FUNCTION_BLOCK CoolingNetwork
VAR_INPUT
	//feed temperature setpoint and system enabling
	fSetPoint_CN : REAL;
	fSetPoint_eChiller : REAL;
	fSetPoint_HVFAStorage : REAL;
	bLoading_HVFAStorage : BOOL;
	bSetStatusOn_eChiller : BOOL;
	bSetStatusOn_HeatPump : BOOL;
	bSetStatusOn_HVFAStorage : BOOL;	
END_VAR
VAR_OUTPUT
	//temperatures in buffer storage
	fTemperatureBufferStorage : REAL;
END_VAR
VAR
	//default parameters
	ST_HVFADefaultParameters : ST_HVFASystemDefaultParameters := (aSetPointLimitsTemperature:=[5,25]);

	//systems
	BufferStorage : FB_BufferStorage;
	eChillerSystem : FB_eChillerSystem;
	HVFAStorage_796 : FB_HVFASystem := (ST_DefaultParameters := ST_HVFADefaultParameters);
	HVFAStorage_795 : FB_HVFAStorage;
	HeatPumpSystem : FB_HeatPumpSystem;
	
	//internal variables
	fAlgorithmPermissionTemperatureRange : REAL := 10; //algorithm mode is only allowed if temperature is between +- 5 K around fSetPointTemperature
	bAlgorithmPermission : BOOL := TRUE;	
END_VAR

//check for algorithm permission
bAlgorithmPermission := Limiter(fInput := BufferStorage.MidTemperature,
								fLowerLimit := fSetPoint_CN-fAlgorithmPermissionTemperatureRange/2,
								fUpperLimit := fSetPoint_CN+fAlgorithmPermissionTemperatureRange);

//buffer storage system
BufferStorage();
fTemperatureBufferStorage := BufferStorage.MidTemperature;

//producer
eChillerSystem(bSetStatusOnAutomatic := bSetStatusOn_eChiller,
	bAlgorithmPermission := bAlgorithmPermission,
	fSetPointAutomatic := fSetPoint_eChiller,
	fExternalTemperature := BufferStorage.MidTemperature);

//NOTE: heat pump systems contains only two-point actors -> fSetPointAutomatic = 0	
HeatPumpSystem(bSetStatusOnAutomatic := bSetStatusOn_HeatPump,
	bAlgorithmPermission := bAlgorithmPermission,
	fSetPointAutomatic := 0);
	
//external storages with pumps 796
HVFAStorage_796(bSetStatusOnAutomatic := bSetStatusOn_HVFAStorage,
	bAlgorithmPermission := bAlgorithmPermission,
	fSetPointAutomatic := fSetPoint_HVFAStorage,
	bLoading := bLoading_HVFAStorage);
	
//external storage without pumps 795
HVFAStorage_795();

END_FUNCTION_BLOCK

(* stored: Version 1.1.0.1, ProductVersion 3.1.4024.10
   POU CoolingNetwork: Id {3e3c7edc-aa3e-40d5-adb7-105c87a52325}, SpecialFunc None *)
